FUNCTION_BLOCK FB_MoverX IMPLEMENTS IMover
VAR
	_id       : UDINT;
	_axisRef  : REFERENCE TO AXIS_REF;
	_position : LREAL;
	_velocity : LREAL;
	_status	: INT;
	_posId	: UDINT;	
END_VAR

METHOD AssignAxisRef : BOOL
VAR_INPUT
	axis	: REFERENCE TO AXIS_REF;
END_VAR
_axisRef REF= axis;
AssignAxisRef := TRUE;
END_METHOD

METHOD AssignID : BOOL
VAR_INPUT
	ID	: UDINT;
END_VAR
_id := ID;
END_METHOD

METHOD GetPosition : LREAL
GetPosition := _position;
END_METHOD

METHOD GetStatus : INT
GetStatus := _status;
END_METHOD

METHOD SetPositionID : BOOL
VAR_INPUT
	ID	: UDINT;
END_VAR
_posId := ID;
END_METHOD

METHOD SetStatus : BOOL
VAR_INPUT
	status	: INT;
END_VAR
_status := status;
SetStatus := true;
END_METHOD

METHOD UpdateData : ST_MoverData
_position := _axisRef.NcToPlc.ModuloActPos;
UpdateData.id := _id;
UpdateData.pos := _position;
UpdateData.status := _status;
UpdateData.assigned := _posId <> 0;
END_METHOD

METHOD UpdatePosition : BOOL
_position := _axisRef.NcToPlc.ModuloActPos;
END_METHOD

END_FUNCTION_BLOCK

(* stored: Version 1.1.0.1, ProductVersion 3.1.4026.12
   POU FB_MoverX: Id {5a7cf214-71b7-4c8d-a77d-204028ecb287}, SpecialFunc None
   Method AssignAxisRef: Id {e1d82af4-8f6a-4c7f-9d48-719d7962cec7}
   Method AssignID: Id {aefc784f-4d23-4fb9-8518-4b089e31af57}
   Method GetPosition: Id {1be03cfb-a6c3-4443-9902-40f951285a9f}
   Method GetStatus: Id {b297532d-4480-4f71-9b83-39026a310b3a}
   Method SetPositionID: Id {6fab7301-0c9c-44e8-9e1d-d609bbb7c89e}
   Method SetStatus: Id {0a7191fb-5e77-4dea-a05d-a0bdca83c510}
   Method UpdateData: Id {7fc6b7f0-a1ce-46fa-a182-acb29a577add}
   Method UpdatePosition: Id {ab62045e-375f-46d3-b7af-e566298d2bb8} *)
